(* CoDeSys 2.3.9.31 project: CL13-ARM.pro *)
(* Libraries: TcBase.lib 14.5.09 11:14:08, TcSystem.lib 27.2.12 14:08:36, TcUtilities.lib 10.1.13 19:12:12, STANDARD.LIB 5.6.98 11:03:02, TcBABasic.lib 29.10.09 13:26:44 *)

(* Task configuration *)
TASK Standard (PRIORITY := 0, INTERVAL := T#10ms);
	MAIN
END_TASK

(* Global variable list: Global_Variables *)
VAR_GLOBAL
	AllLightsOn: BOOL;
	AllLightsOff: BOOL;

	IsAllesUitInAchterbouw : BOOL; (* feedback over lichtstatus achterbouw *)
	IsAllesUitInSalon : BOOL; (* feedback over lichtstatus salon *)

	LED_Rolluik_Voorgevel_Up AT %Q*: BOOL;  (*Terugkoppeling status neersignaal*)
	LED_Rolluik_Voorgevel_Down AT %Q*: BOOL; (*Terugkoppeling status neersignaal*)

	(* Tijdsgerelateerde zaken *)
	time_RTC 				: DT;
	time_RTCEX 				: DT;
	time_RTCEX2 			: TIMESTRUCT;
	nMicroseconds 			: DWORD;

	firstCycle					: BOOL;
	status 					: StatusVariables;
	WaterTeller				:UDINT;
	AutoMode				: BOOL;
END_VAR

(* Global variable list: Input_variables *)
VAR_GLOBAL
	DK_Gang_A AT %I*: BOOL;
	DK_Gang_B AT %I*: BOOL;
	DK_Gang_C AT %I*: BOOL;
	DK_Gang_D AT %I*: BOOL;
	DK_Voordeur_BEL AT %I*: BOOL;
	DK_Toilet AT %I*:BOOL;

(* D1 / centrale kolom keuken - 1 / 6V*)
	DK_Kolom1_A  AT %I*: BOOL; (* Eiland *)
	DK_Kolom1_B  AT %I*: BOOL; (* Eettafel DIMMER *)
	DK_Kolom1_C  AT %I*: BOOL; (* Waskot *)
	DK_Kolom1_D  AT %I*: BOOL; (* Grid IN - Bureau *)
	DK_Kolom1_E  AT %I*: BOOL; (* Dampkap *)
	DK_Kolom1_F  AT %I*: BOOL; (*  *)

(* D2 / centrale kolom keuken - 2 / 4V*)
	DK_Kolom2_A  AT %I*: BOOL; (* Renson Eco *)
	DK_Kolom2_B  AT %I*: BOOL; (* Renson HDC *)
	DK_Kolom2_C  AT %I*: BOOL; (* Renson Boost/Nightcooling *)
	DK_Kolom2_D  AT %I*: BOOL; (* Renson Empty House *)

(* D3 / achtergevel - 1 / 6V*)
	DK_Achtergevel_A  AT %I*: BOOL; (* Buitenverlichting *)
	DK_Achtergevel_B  AT %I*: BOOL; (* Eettafel DIMMER *)
	DK_Achtergevel_C  AT %I*: BOOL; (* Ontbijtkast *)
	DK_Achtergevel_D  AT %I*: BOOL; (*  *)
	DK_Achtergevel_E  AT %I*: BOOL; (* Rolgordijn op *)
	DK_Achtergevel_F  AT %I*: BOOL; (* Rolgordijn neer  *)

(* D11 / Salon / 4V *)
	DK_Salon_A  AT %I*: BOOL; (* Wandlampen zetel DIMMER *)
	DK_Salon_B  AT %I*: BOOL; (*  Rolluik voorgevel *)
	DK_Salon_C  AT %I*: BOOL; (*  *)
	DK_Salon_D  AT %I*: BOOL; (*  *)

	NC_Water AT %I*:BOOL; (* NC contact Elster watermeter *)

END_VAR

(* Global variable list: Output_variables *)
VAR_GLOBAL
	L1_Oversteek 	AT %Q* 		: BOOL; 	(* Oversteek buiten *)
	L2_Eettafel		AT %Q* 		: UINT; 	(* Licht boven de eettafel *)
	L3_Bureau		AT %Q* 		: BOOL;	(* Licht bureau *)
	L4_Ontbijtkast 	AT %Q*		: BOOL;
	L5_Eiland		AT %Q* 		: BOOL; 	(* L5 - Deltalight profiel boven eiland *)
	L6_Bijkeuken		AT %Q*		: BOOL;	(* verlichting in de bijkeuken *)
	L7_Living		AT %Q* 		: BOOL; 	(* Licht living *)
	L8_Salon		AT %Q*		: UINT; 	(* Licht salon *)

	L_Gang_GLV 		AT %Q* 		: BOOL; 	(* L10 *)
	L_Toilet 			AT %Q* 		: BOOL;    (* L11 *)
	L_Kelder 		AT %Q* 		: BOOL;    (* L12_Licht kelder *)

	L2_Status 					: BOOL; 	(* Terugkoppeling van de status voor het licht boven de eettafel *)
	L8_Status 					: BOOL; 	(* Terugkoppeling van de status voor het licht in het salon *)


	HealthBox 		AT %Q* 		: BOOL; (* 230v Renson Healthbox *)
	DK_Kolom1_LED 	AT %Q* 		: BOOL;
	DK_Salon_LED 	AT %Q*		 : BOOL;
	DK_Kolom2_LED1 AT %Q*		 : BOOL;
	DK_Achtergevel_LED AT %Q* 	: BOOL;

	Auto_Rolluik_Voorgevel_Up	: BOOL;
	Auto_Rolluik_Voorgevel_Down	: BOOL;



	Rolluik_Voorgevel_Up AT %Q* : BOOL;
	Rolluik_Voorgevel_Down AT %Q* : BOOL;
	Deurbel AT %Q* : BOOL;

	M_Keuken_Op 		AT %Q* 		: BOOL;
	M_Keuken_Neer		AT %Q*		: BOOL;

(* een bit wordt geadresseerd door middel van een "Byte nr"."Bit nr"
Waarbij de byte nummer gewoon mag optellen en de bitnummer gaat van 0 tot en met 7 *)

	(*merker_OmTeTesten	AT %MX0.0 : BOOL;
	M_Licht_Eiland		AT %MX0.1 : BOOL;*)

END_VAR

(* Global variable list: PushButtons *)
VAR_GLOBAL

	Button_Kolom1_A : FB_Click;
	Button_Kolom1_C: FB_Click;
	Button_Kolom1_D: FB_Click;
	Button_Kolom1_E: FB_Click;
	Button_Kolom1_F: FB_Click;

	Click_Kolom2_A: FB_Click;
	Click_Kolom2_B: FB_Click;
	Click_Kolom2_C: FB_Click;
	Click_Kolom2_D: FB_Click;

	Click_Toilet : FB_Click;
	Click_Salon_A : FB_Click;
	Click_Salon_B : FB_Click;
	Click_Salon_C : FB_Click;
	Click_Salon_D: FB_Click;

	PushButton_Gang_A: FB_Toggle;
	PushButton_Gang_B: FB_Click;
	PushButton_Gang_C: FB_Toggle;
	PushButton_Gang_D: FB_Click;

	PushButton_Achtergevel_A : FB_Click;
	PushButton_Achtergevel_B : FB_Click;
	PushButton_Achtergevel_C: FB_Click;
	PushButton_Achtergevel_D: FB_Click;
	PushButton_Achtergevel_E: FB_Click;
	PushButton_Achtergevel_F: FB_Click;


END_VAR

(* Global variable list: TwinCAT_Configuration *)
(* Generated automatically by TwinCAT - (read only) *)
VAR_CONFIG
	.LED_Rolluik_Voorgevel_Up AT %QX4.0 : BOOL;
	.LED_Rolluik_Voorgevel_Down AT %QX4.1 : BOOL;
	.DK_Gang_A AT %IX0.0 : BOOL;	(*  ~ {LinkedWith:TIID^Device 2 (CX8000-BK)^Box 1 (CX8000-BK)^Term 2 (KL1859)^Channel 1^Input} *)
	.DK_Gang_B AT %IX0.1 : BOOL;	(*  ~ {LinkedWith:TIID^Device 2 (CX8000-BK)^Box 1 (CX8000-BK)^Term 2 (KL1859)^Channel 2^Input} *)
	.DK_Gang_C AT %IX0.2 : BOOL;	(*  ~ {LinkedWith:TIID^Device 2 (CX8000-BK)^Box 1 (CX8000-BK)^Term 2 (KL1859)^Channel 3^Input} *)
	.DK_Gang_D AT %IX0.3 : BOOL;	(*  ~ {LinkedWith:TIID^Device 2 (CX8000-BK)^Box 1 (CX8000-BK)^Term 2 (KL1859)^Channel 4^Input} *)
	.DK_Voordeur_BEL AT %IX0.4 : BOOL;	(*  ~ {LinkedWith:TIID^Device 2 (CX8000-BK)^Box 1 (CX8000-BK)^Term 2 (KL1859)^Channel 6^Input} *)
	.DK_Toilet AT %IX0.5 : BOOL;	(*  ~ {LinkedWith:TIID^Device 2 (CX8000-BK)^Box 1 (CX8000-BK)^Term 2 (KL1859)^Channel 5^Input} *)
	.DK_Kolom1_A AT %IX0.6 : BOOL;	(*  ~ {LinkedWith:TIID^Device 2 (CX8000-BK)^Box 1 (CX8000-BK)^Term 3 (KL1809)^Channel 1^Input} *)
	.DK_Kolom1_B AT %IX0.7 : BOOL;	(*  ~ {LinkedWith:TIID^Device 2 (CX8000-BK)^Box 1 (CX8000-BK)^Term 3 (KL1809)^Channel 2^Input} *)
	.DK_Kolom1_C AT %IX1.0 : BOOL;	(*  ~ {LinkedWith:TIID^Device 2 (CX8000-BK)^Box 1 (CX8000-BK)^Term 3 (KL1809)^Channel 3^Input} *)
	.DK_Kolom1_D AT %IX1.1 : BOOL;	(*  ~ {LinkedWith:TIID^Device 2 (CX8000-BK)^Box 1 (CX8000-BK)^Term 3 (KL1809)^Channel 4^Input} *)
	.DK_Kolom1_E AT %IX1.2 : BOOL;	(*  ~ {LinkedWith:TIID^Device 2 (CX8000-BK)^Box 1 (CX8000-BK)^Term 3 (KL1809)^Channel 5^Input} *)
	.DK_Kolom1_F AT %IX1.3 : BOOL;	(*  ~ {LinkedWith:TIID^Device 2 (CX8000-BK)^Box 1 (CX8000-BK)^Term 3 (KL1809)^Channel 6^Input} *)
	.DK_Kolom2_A AT %IX1.4 : BOOL;
	.DK_Kolom2_B AT %IX1.5 : BOOL;
	.DK_Kolom2_C AT %IX1.6 : BOOL;
	.DK_Kolom2_D AT %IX1.7 : BOOL;
	.DK_Achtergevel_A AT %IX8.0 : BOOL;	(*  ~ {LinkedWith:TIID^Device 2 (CX8000-BK)^Box 1 (CX8000-BK)^Term 3 (KL1809)^Channel 11^Input} *)
	.DK_Achtergevel_B AT %IX8.1 : BOOL;	(*  ~ {LinkedWith:TIID^Device 2 (CX8000-BK)^Box 1 (CX8000-BK)^Term 3 (KL1809)^Channel 12^Input} *)
	.DK_Achtergevel_C AT %IX8.2 : BOOL;	(*  ~ {LinkedWith:TIID^Device 2 (CX8000-BK)^Box 1 (CX8000-BK)^Term 3 (KL1809)^Channel 13^Input} *)
	.DK_Achtergevel_D AT %IX8.3 : BOOL;	(*  ~ {LinkedWith:TIID^Device 2 (CX8000-BK)^Box 1 (CX8000-BK)^Term 3 (KL1809)^Channel 14^Input} *)
	.DK_Achtergevel_E AT %IX8.4 : BOOL;	(*  ~ {LinkedWith:TIID^Device 2 (CX8000-BK)^Box 1 (CX8000-BK)^Term 3 (KL1809)^Channel 15^Input} *)
	.DK_Achtergevel_F AT %IX8.5 : BOOL;	(*  ~ {LinkedWith:TIID^Device 2 (CX8000-BK)^Box 1 (CX8000-BK)^Term 3 (KL1809)^Channel 16^Input} *)
	.DK_Salon_A AT %IX2.0 : BOOL;	(*  ~ {LinkedWith:TIID^Device 2 (CX8000-BK)^Box 1 (CX8000-BK)^Term 3 (KL1809)^Channel 7^Input} *)
	.DK_Salon_B AT %IX2.1 : BOOL;	(*  ~ {LinkedWith:TIID^Device 2 (CX8000-BK)^Box 1 (CX8000-BK)^Term 3 (KL1809)^Channel 8^Input} *)
	.DK_Salon_C AT %IX2.2 : BOOL;	(*  ~ {LinkedWith:TIID^Device 2 (CX8000-BK)^Box 1 (CX8000-BK)^Term 3 (KL1809)^Channel 9^Input} *)
	.DK_Salon_D AT %IX2.3 : BOOL;	(*  ~ {LinkedWith:TIID^Device 2 (CX8000-BK)^Box 1 (CX8000-BK)^Term 3 (KL1809)^Channel 10^Input} *)
	.NC_Water AT %IX4.0 : BOOL;	(*  ~ {LinkedWith:TIID^Device 2 (CX8000-BK)^Box 1 (CX8000-BK)^Term 5 (KL1809)^Channel 1^Input} *)
	.L1_Oversteek AT %QX20.0 : BOOL;	(*  ~ {LinkedWith:TIID^Device 2 (CX8000-BK)^Box 1 (CX8000-BK)^Term 6 (KL2809)^Channel 1^Output} *)
	.L2_Eettafel AT %QB16 : UINT;	(*  ~ {LinkedWith:TIID^Device 2 (CX8000-BK)^Box 1 (CX8000-BK)^Term 13 (KL2751)^Channel 1^Data Out} *)
	.L3_Bureau AT %QX20.1 : BOOL;	(*  ~ {LinkedWith:TIID^Device 2 (CX8000-BK)^Box 1 (CX8000-BK)^Term 6 (KL2809)^Channel 2^Output} *)
	.L4_Ontbijtkast AT %QX20.2 : BOOL;
	.L5_Eiland AT %QX20.3 : BOOL;
	.L6_Bijkeuken AT %QX20.4 : BOOL;
	.L7_Living AT %QX20.5 : BOOL;
	.L8_Salon AT %QB18 : UINT;	(*  ~ {LinkedWith:TIID^Device 2 (CX8000-BK)^Box 1 (CX8000-BK)^Term 14 (KL2751)^Channel 1^Data Out} *)
	.L_Gang_GLV AT %QX4.5 : BOOL;	(*  ~ {LinkedWith:TIID^Device 2 (CX8000-BK)^Box 1 (CX8000-BK)^Term 6 (KL2809)^Channel 14^Output} *)
	.L_Toilet AT %QX4.6 : BOOL;	(*  ~ {LinkedWith:TIID^Device 2 (CX8000-BK)^Box 1 (CX8000-BK)^Term 6 (KL2809)^Channel 13^Output} *)
	.L_Kelder AT %QX4.4 : BOOL;	(*  ~ {LinkedWith:TIID^Device 2 (CX8000-BK)^Box 1 (CX8000-BK)^Term 6 (KL2809)^Channel 16^Output} *)
	.HealthBox AT %QX5.5 : BOOL;	(*  ~ {LinkedWith:TIID^Device 2 (CX8000-BK)^Box 1 (CX8000-BK)^Term 2 (KL1859)^Channel 8^Output} *)
	.DK_Kolom1_LED AT %QX5.6 : BOOL;	(*  ~ {LinkedWith:TIID^Device 2 (CX8000-BK)^Box 1 (CX8000-BK)^Term 7 (KL2809)^Channel 2^Output} *)
	.DK_Salon_LED AT %QX5.7 : BOOL;	(*  ~ {LinkedWith:TIID^Device 2 (CX8000-BK)^Box 1 (CX8000-BK)^Term 7 (KL2809)^Channel 1^Output} *)
	.DK_Kolom2_LED1 AT %QX6.0 : BOOL;
	.DK_Achtergevel_LED AT %QX20.6 : BOOL;
	.Rolluik_Voorgevel_Up AT %QX5.0 : BOOL;	(*  ~ {LinkedWith:TIID^Device 2 (CX8000-BK)^Box 1 (CX8000-BK)^Term 8 (KL2012)^Channel 1^Output} *)
	.Rolluik_Voorgevel_Down AT %QX5.1 : BOOL;	(*  ~ {LinkedWith:TIID^Device 2 (CX8000-BK)^Box 1 (CX8000-BK)^Term 8 (KL2012)^Channel 2^Output} *)
	.Deurbel AT %QX5.2 : BOOL;	(*  ~ {LinkedWith:TIID^Device 2 (CX8000-BK)^Box 1 (CX8000-BK)^Term 2 (KL1859)^Channel 4^Output} *)
	.M_Keuken_Op AT %QX12.1 : BOOL;	(*  ~ {LinkedWith:TIID^Device 2 (CX8000-BK)^Box 1 (CX8000-BK)^Term 9 (KL2012)^Channel 1^Output} *)
	.M_Keuken_Neer AT %QX12.2 : BOOL;	(*  ~ {LinkedWith:TIID^Device 2 (CX8000-BK)^Box 1 (CX8000-BK)^Term 9 (KL2012)^Channel 2^Output} *)
END_VAR

(* Global variable list: Visualisation_variables *)
VAR_GLOBAL

	Visu_Licht_Oversteek		AT %MX0.0 			: BOOL;
	Visu_Dimmer_Eettafel		AT %MX0.1 			: BOOL;
	Visu_L3 					AT %MX0.2			: BOOL; (* Licht bureau *)
	Visu_Ontbijtkast 			AT %MX0.3			: BOOL;
	Visu_Eiland				AT %MX0.4			: BOOL;
	Visu_Bijkeuken			AT %MX0.5			: BOOL;
	Visu_Licht_Living 			AT %MX0.6			: BOOL;
	Visu_Dimmer_Salon 		AT %MX0.7 			: BOOL;

	Visu_Salon_TV			AT %MX0.8			: BOOL; (* Nog niet in gebruik *)
	Visu_Licht_Gang			AT %MX0.9			: BOOL; (* L10 *)
	Visu_Licht_Toilet 			AT %MX0.10			: BOOL; (* L11 *)
	Visu_Licht_Kelder			AT %MX0.11			: BOOL; (* L12 *)

	(* Andere lichten komen hier *)

	Visu_Rolluik_Voorgevel_Up	AT %MX2.0	 	: BOOL;
	Visu_Rolluik_Voorgevel_Down	AT %MX2.1	 	: BOOL;
	Visu_Rolgordijn_Up			AT %MX2.3		: BOOL;
	Visu_Rolgordijn_Neer			AT %MX2.4		: BOOL;
	Visu_AllesUit 					AT %MX2.5		: BOOL;

	Visu_Deurbel 				: BOOL;
	Visu_AllesAan 				: BOOL;
	Visu_HEALTHBOX			: BOOL; (* Healthbox *)
	Visu_Dimmer_Salon_Status		: REAL;
	Visu_Dimmer_Eettafel_Status	: REAL;

	Visu_Sfeer_Avond				: BOOL;
	Visu_AutoMode				: BOOL;


(* alle types die op een byte grootte hebben, woorden weergegeven zoals:
	MerkerByte_2		AT %MB2 : BYTE;
	MerkerByte_3		AT %MB3 : BYTE;
	MerkerByte_4		AT %MB4 : BYTE;
	MerkerByte_5		AT %MB5 : BYTE;

(* alle types die op een woord grootte hebben, woorden weergegeven zoals: *)
	MerkerWoord_10		AT %MW10 : INT;
	MerkerWoord_12		AT %MW12 : UINT;
	MerkerWoord_14		AT %MW14 : INT;
	MerkerWoord_16		AT %MW16 : UINT;

(* alle types die op een dubbelwoord grootte hebben, woorden weergegeven zoals: *)
	MerkerDWoord_20		AT %MD20 : DINT;
	MerkerDWoord_24		AT %MD24 : UDINT;
	MerkerDWoord_28		AT %MD28 : REAL;
	MerkerDWoord_32		AT %MD32 : UINT;

*)


END_VAR

(* Data type *)
TYPE StatusVariables :
STRUCT

END_STRUCT
END_TYPE

(* POU MAIN, ST *)
PROGRAM MAIN
VAR
END_VAR
Process_Inputs;
Rolluiken;
Deurbel_Programma;
Dimmers;
Control_Lights_ST;
Ventilation;
BezorgFeedbackAanLeds;
PRG_Clock;
MAIN_1;

firstCycle := Systemtaskinfoarr[1].firstCycle;
(*SetStatusStruct; *)
Smartmeters;
ResetInputs;
END_PROGRAM

(* POU Process_Inputs, ST *)
PROGRAM Process_Inputs
VAR
	R_Trig_AllesUit: R_TRIG;
END_VAR
PushButton_Gang_B(ingang:= DK_Gang_B); (* linkt de fysieke input aan de functie block FB_Click *)
PushButton_Gang_D(ingang:= DK_Gang_D);
Button_Kolom1_A(ingang:= DK_Kolom1_A);
Button_Kolom1_C(ingang:= DK_Kolom1_C);
Button_Kolom1_D(ingang:= DK_Kolom1_D);
Button_Kolom1_E(ingang:= DK_Kolom1_E);
Button_Kolom1_F(ingang:= DK_Kolom1_F);
Click_Toilet(ingang:= DK_Toilet);

Click_Kolom2_A(ingang := DK_Kolom2_A);
Click_Kolom2_B(ingang := DK_Kolom2_B);
Click_Kolom2_C(ingang := DK_Kolom2_C);
Click_Kolom2_D(ingang := DK_Kolom2_D);

PushButton_Achtergevel_A(ingang:= DK_Achtergevel_A);
PushButton_Achtergevel_B(ingang:= DK_Achtergevel_B);
PushButton_Achtergevel_C(ingang:= DK_Achtergevel_C);
PushButton_Achtergevel_D(ingang:= DK_Achtergevel_D);
PushButton_Achtergevel_E(ingang:= DK_Achtergevel_E);
PushButton_Achtergevel_F(ingang:= DK_Achtergevel_F);

AllLightsOff := Visu_AllesUit OR PushButton_Gang_D.LangClick;
AllLightsOn := Visu_AllesAan OR PushButton_Gang_D.TweeClick;
END_PROGRAM

(* POU Rolluiken, ST *)
PROGRAM Rolluiken
VAR
	Rolluik_Voorgevel: Rolluik;
	Rolgordijn_Keuken: Rolluik;
END_VAR
Rolgordijn_Keuken
(
	DrukknopOp:=  PushButton_Achtergevel_D.EenClick OR Visu_Rolgordijn_Up,
	DrukknopNeer:= PushButton_Achtergevel_C.EenClick OR Visu_Rolgordijn_Neer,
	Tijd:= t#100s,
	UitgOp=> M_Keuken_Op,
	UitgNeer=>M_Keuken_Neer );

Rolluik_Voorgevel
(
	DrukknopOp:=  Button_Kolom1_D.EenClick OR Visu_Rolluik_Voorgevel_Up OR Click_Salon_D.EenClick,
	DrukknopNeer:= Button_Kolom1_C.EenClick OR Visu_Rolluik_Voorgevel_Down OR Click_Salon_C.TweeClick,
	Tijd:= t#20s,
	UitgOp=> Rolluik_Voorgevel_Up,
	UitgNeer=>Rolluik_Voorgevel_Down );
END_PROGRAM

(* POU TestCode/Rolluik, ST *)
FUNCTION_BLOCK Rolluik
VAR_INPUT
	DrukknopOp: BOOL;
	DrukknopNeer: BOOL;
	Tijd: TIME := t#20s;
END_VAR
VAR_OUTPUT
	UitgOp: BOOL;
	UitgNeer: BOOL;
END_VAR
VAR
	Stap: INT;
	TimerOp: TON;
	TimerNeer: TON;
	rDrukknopOp: R_TRIG;
	rDrukknopNeer: R_TRIG;
END_VAR
TimerOp(IN:= Stap = 10 , PT:= Tijd , Q=> , ET=> );
TimerNeer(IN:= Stap = 20 , PT:= Tijd , Q=> , ET=> );

rDrukknopOp(CLK:= DrukknopOp , Q=> );
rDrukknopNeer(CLK:= DrukknopNeer , Q=> );

CASE Stap OF

0:
	IF rDrukknopOp.Q THEN
		Stap := 10;
	END_IF

	IF rDrukknopNeer.Q THEN
		Stap := 20;
	END_IF

10:
	IF DrukknopNeer OR TimerOp.Q  THEN
		Stap := 0;
	END_IF

20:

	IF DrukknopOp OR TimerNeer.Q THEN
		Stap := 0;
	END_IF

END_CASE


UitgOp := Stap = 10;
UitgNeer := Stap = 20;
END_FUNCTION_BLOCK

(* POU Deurbel_Programma, LD *)
PROGRAM Deurbel_Programma
VAR
	Timer_Deurbel: TOF;
	Status_Deurbel: BOOL;
END_VAR
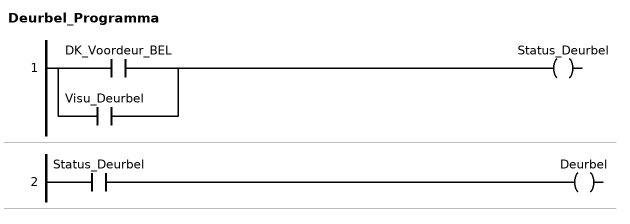
_LD_ (* Ladder Diagram *)
NETWORK 1
	{ [DK_Voordeur_BEL] | [Visu_Deurbel] } --- (Status_Deurbel)
NETWORK 2
	[Status_Deurbel] --- (Deurbel)
_END_LD_
(* the same logic as Structured Text *)
(* Network 1 *)
Status_Deurbel := DK_Voordeur_BEL OR Visu_Deurbel;
(* Network 2 *)
Deurbel := Status_Deurbel;
END_PROGRAM

(* POU Dimmers, ST *)
PROGRAM Dimmers
VAR
	Dimmer_Eettafel: FB_Dimmer1SwitchEco;
	(*Dimmer_Eettafel2: FB_Dimmer1Switch;*)
	Dimmer_SalonL9: FB_Dimmer1SwitchEco;
END_VAR
Dimmer_Eettafel
(
bSwitchDimm:= Visu_Dimmer_Eettafel OR PushButton_Gang_B.TweeClick OR DK_Kolom1_B,
tDimmTime:= t#3s,
bOn:= AllLightsOn,
bOff:= AllLightsOff,
nOut=>L2_Eettafel,
bLight => L2_Status,
);

Visu_Dimmer_Salon_Status := OnAScaleOfZeroToTen(L8_Salon);
Visu_Dimmer_Eettafel_Status := OnAScaleOfZeroToTen(L2_Eettafel);

Dimmer_SalonL9
(
	bSwitchDimm:= DK_Salon_A OR Visu_Dimmer_Salon,
	bOn:= AllLightsOn,
	bOff:= AllLightsOff,
	tSwitchOverTime:= ,
	tDimmTime:= t#3s,

	nOut=>L8_Salon ,
	bLight=>L8_Status );
END_PROGRAM

(* POU Functions/OnAScaleOfZeroToTen, ST *)
FUNCTION OnAScaleOfZeroToTen : LREAL
VAR_INPUT
	ValueIn : INT;

END_VAR
VAR
END_VAR
OnAScaleOfZeroToTen := ValueIn /  3267.6;
END_FUNCTION

(* POU Control_Lights_ST, ST *)
PROGRAM Control_Lights_ST
VAR
	FB_Light_Hallway_Downstairs: FB_Light;
	FB_Light_Toilet: FB_Light;
	FB_Light_3: FB_Light;
	FB_Light_Oversteek: FB_Light;
	FB_Light_Ontbijtkast: FB_Light;
	FB_Light_Eiland : FB_Light;
	FB_Light_Kelder : FB_Light;
	FB_Light_Wasplaats : FB_Light;
	FB_Sfeer_Avond_Salon : FB_Sfeer;

	FB_Light_Living: FB_Light;
	FB_Auto_Mode: FB_Light;
END_VAR
FB_Light_Hallway_Downstairs(
	bOn:= AllLightsOn ,
	bOff:=AllLightsOff ,
	bToggle:= Visu_Licht_Gang OR DK_Gang_C
	 , bLight=> L_Gang_GLV);

FB_Auto_Mode(
	bOn:= 0 ,
	bOff:=0 ,
	bToggle:=Click_Toilet.LangClick OR Visu_AutoMode
	 , bLight=> AutoMode);

FB_Light_Toilet(
	bOn:= 0 ,
	bOff:=AllLightsOff ,
	bToggle:=Visu_Licht_Toilet OR Click_Toilet.EenClick
	 , bLight=> L_Toilet);

FB_Light_3(
	bOn:= AllLightsOn ,
	bOff:=AllLightsOff ,
	bToggle:=Button_Kolom1_A.TweeClick OR Visu_L3
	 , bLight=> L3_Bureau);

FB_Light_Oversteek(
	bOn:= 0 ,
	bOff:=AllLightsOff ,
	bToggle:=Visu_Licht_Oversteek OR PushButton_Achtergevel_A.EenClick
	 , bLight=> L1_Oversteek);

FB_Light_Ontbijtkast(
	bOn := AllLightsOn,
	bOff := AllLightsOff,
	bToggle := PushButton_Achtergevel_B.EenClick OR Visu_Ontbijtkast,
	bLight => L4_Ontbijtkast);

FB_Light_Eiland(
	bOn := AllLightsOn,
	bOff := AllLightsOff,
	bToggle := Button_Kolom1_A.EenClick OR Visu_Eiland,
	bLight => L5_Eiland);

FB_Light_Kelder(
	bOn := 0,
	bOff := AllLightsOff,
	bToggle := PushButton_Gang_B.EenClick OR Visu_Licht_Kelder,
	bLight => L_Kelder);


FB_Light_Wasplaats(
	bOn := AllLightsOn,
	bOff := AllLightsOff,
	bToggle := Button_Kolom1_E.EenClick OR Visu_Bijkeuken,
	bLight => L6_Bijkeuken);

FB_Light_Living
(
	bOn :=AllLightsOn,
	bOff := AllLightsOff,
	bToggle := Button_Kolom1_F.EenClick OR Visu_Licht_Living,
	bLight => L7_Living);

(* FB_Sfeer_Avond_Salon(Trigger:= Visu_Sfeer_Avond, default:= 0, Uitgang => L3_Bureau);*)
END_PROGRAM

(* POU TestCode/FB_Sfeer, ST *)
FUNCTION_BLOCK FB_Sfeer
VAR_INPUT
	Trigger : BOOL;
	default: BOOL;
END_VAR
VAR_OUTPUT
	Uitgang : BOOL;
END_VAR
VAR
	Getriggerd: R_TRIG;
	DoUwDing: BOOL;
END_VAR
Getriggerd(CLK:= Trigger, Q => DoUwDing);

IF DoUwDing THEN
	Uitgang := default;
END_IF
END_FUNCTION_BLOCK

(* POU Ventilation, ST *)
PROGRAM Ventilation
VAR
	FB_Ventilation_OnOff: FB_Light;
END_VAR
FB_Ventilation_OnOff(
	bOn:= 0 ,
	bOff:=0 ,
	bToggle:= Visu_HealthBox OR Button_Kolom1_E.LangClick
	 , bLight=> HealthBox);
END_PROGRAM

(* POU BezorgFeedbackAanLeds, ST *)
PROGRAM BezorgFeedbackAanLeds
VAR
END_VAR
DK_Kolom1_LED :=	NOT L5_Eiland
					AND NOT L2_Status
					AND NOT L3_Bureau
					AND NOT AutoMode;

DK_Achtergevel_LED := DK_Kolom1_LED;

DK_Salon_LED := 		NOT L8_Status AND NOT AutoMode;

DK_Kolom2_LED1 := HealthBox;
END_PROGRAM

(* POU PRG_Clock, ST *)
PROGRAM PRG_Clock
VAR
	NT_GetTime_CX				: NT_GetTime;
	GetTime						: DT;
	Clock						: RTC;

	PC_Clock_Valid				: BOOL;
	RTC_Clock_Valid				: BOOL;

	Actual_Time 					: TOD;
	Actual_Date 					: DATE;

	Actual_Date_Time				: STRING;

	Actual_Hour					: WORD;
	Actual_Minute					: WORD;
	Actual_Second				: WORD;
	Actual_Year					: WORD;
	Actual_Month					: WORD;
	Actual_Day					: WORD;
END_VAR
(* Bios time and date from PC or CX *)
NT_GetTime_CX(
	NETID		:= 	'200.255.255.154.1.1',									(* AMS NetID from PC or CX, empty string is lokal *)
	START		:= 	SystemTaskInfoArr[1].firstCycle OR						(* Update after start Runtime *)
					(DT_TO_TOD(Clock.CDT)=TOD#00:00:00) OR				(* Update if 'Clock' empty *)
					MID(DT_TO_STRING(Clock.CDT),2,21)='00',				(* Update each minute *)
	TMOUT		:= 	t#1s ,
	 );

PC_Clock_Valid 	:= NOT NT_GetTime_CX.BUSY AND NOT NT_GetTime_CX.START;

(* Time from external device *)
IF PC_Clock_Valid THEN
	GetTime := SYSTEMTIME_TO_DT(NT_GetTime_CX.TIMESTR);
END_IF

Clock(																	(* Internal clock, independent with Windows clock *)
	EN			:= PC_Clock_Valid,
	PDT		:= GetTime
	 );

RTC_Clock_Valid	:= Clock.Q;

(* Date en Time *)
IF RTC_Clock_Valid THEN
	Actual_Time 				:= DT_TO_TOD(Clock.CDT);
	Actual_Date				:= DT_TO_DATE(Clock.CDT);

	Actual_Date_Time			:= DT_TO_STRING(Clock.CDT);

	Actual_Hour 				:= STRING_TO_INT(MID(Actual_Date_Time,2,15));
	Actual_Minute 			:= STRING_TO_INT(MID(Actual_Date_Time,2,18));
	Actual_Second 			:= STRING_TO_INT(MID(Actual_Date_Time,2,21));
	Actual_Year 				:= STRING_TO_INT(MID(Actual_Date_Time,4,4));
	Actual_Month 				:= STRING_TO_INT(MID(Actual_Date_Time,2,9));
	Actual_Day 				:= STRING_TO_INT(MID(Actual_Date_Time,2,12));
END_IF
END_PROGRAM

(* POU MAIN_1, ST *)
PROGRAM MAIN_1
VAR
	CurrentTime			: TOD;
	tRolluikOp			: TOD;
	tRolluikNeer			: TOD;
	tLightGangAan		: TOD;
	tLightGangUit			: TOD;

	tLichtGangAan: TOD;
	tLichtGangUit: TOD;
	tTestAan: TOD;
	tTestUit: TOD;
	strTime: STRING;
END_VAR
P_RTC_ST;

(* dsjkfsjlqfs *)
IF firstCycle	THEN

	tRolluikOp := TOD#07:30:00;
	tRolluikNeer := TOD#17:48:30;

	tLichtGangAan:= TOD#21:04:00;
	tLichtGangUit:= TOD#22:43:00;

	tTestAan	:= TOD#00:00:00;
	tTestUit:= TOD#08:00:00;

END_IF

	tRolluikOp := TOD#07:30:00;
	tRolluikNeer := TOD#17:48:30;

	tLichtGangAan:= TOD#21:04:00;
	tLichtGangUit:= TOD#22:43:00;

	tTestAan	:= TOD#23:58:00;
	tTestUit:= TOD#23:59:00;

CurrentTime := DT_TO_TOD(time_RTC);
strTime := TOD_TO_STRING(CurrentTime);

IF AutoMode THEN
	IF CurrentTime > tRolluikOp AND CurrentTime < tRolluikNeer  THEN
	Rolluik_Voorgevel_Up := TRUE;
	Rolluik_Voorgevel_Down := FALSE;
	ELSE
	Rolluik_Voorgevel_Up := FALSE;
	Rolluik_Voorgevel_Down := TRUE;
	END_IF

	IF CurrentTime > tLichtGangAan AND CurrentTime < tLichtGangUit THEN
	L_Gang_GLV := TRUE;
	ELSE
	L_Gang_GLV := FALSE;
	END_IF
ELSE
;
	(*Rolluik_Voorgevel_Up := FALSE;
	Rolluik_Voorgevel_Down := FALSE;*)
END_IF


(*IF CurrentTime > tTestAan AND CurrentTime < tTestUit THEN
HealthBox := TRUE;
ELSE
HealthBox := FALSE;
END_IF*)
END_PROGRAM

(* POU tcUtilities/Converting/Formatting/P_RTC_ST, ST *)
PROGRAM P_RTC_ST
VAR
	syncTimer 				: TON;
	fbGetLocalTime 			: NT_GetTime;
	syncTrigger 			: F_TRIG;
	bBusy 					: BOOL;
	bError 					: BOOL;
	nErrID 					: UDINT;
	presetTime 				: TIMESTRUCT;

	fbRTC 					: RTC;
	bValid_RTC 				: BOOL;

	fbRTC_EX 				: RTC_EX;
	bValid_RTCEX 			: BOOL;
	nMilliseconds 			: DWORD;

	fbRTC_EX2 				: RTC_EX2;
	bValid_RTCEX2 			: BOOL;

END_VAR
syncTimer(
	IN			:= NOT syncTimer.q,
	PT			:= T#5s,
	Q			=> ,
	ET			=> );

fbGetLocalTime(
	NETID		:= ,
	START		:= syncTimer.Q	OR systemtaskinfoarr[1].firstCycle,
	TMOUT		:= ,
	BUSY		=> ,
	ERR		=> bError,
	ERRID		=> nErrID,
	TIMESTR	=> presetTime);

syncTrigger(
	CLK			:= fbGetLocalTime.BUSY AND NOT bError,
	Q=> 			);

fbRTC(
	EN			:= syncTrigger.Q,
	PDT		:= SYSTEMTIME_TO_DT(presetTime),
	Q			=> bValid_RTC,
	CDT=> 		time_RTC);

fbRTC_EX(
	EN			:= syncTrigger.Q,
	PDT		:= SYSTEMTIME_TO_DT(presetTime),
	PMSEK		:= presetTime.wMilliseconds,
	Q			=> bValid_RTCEX,
	CDT		=> time_RTCEX,
	CMSEK		=> nMilliseconds);

fbRTC_EX2(
	EN			:= syncTrigger.Q,
	PDT		:= presetTime,
	PMICRO		:= 0,
	Q			=> bValid_RTCEX2,
	CDT		=> time_RTCEX2,
	CMICRO		=> nMicroseconds);
END_PROGRAM

(* POU Smartmeters, ST *)
PROGRAM Smartmeters
VAR
	fet_pulse		: F_TRIG;
	pulse		: BOOL;
	NoChange	: BOOL;
END_VAR
VAR RETAIN PERSISTENT
	teller		: UDINT;
END_VAR
NoChange:= NC_Water;

IF NoChange = TRUE THEN
	pulse:= FALSE;
END_IF

fet_pulse(clk:=NC_Water);
pulse := fet_pulse.Q;

IF pulse THEN
	teller:= teller + 1;
END_IF

WaterTeller:=teller;
END_PROGRAM

(* POU ResetInputs, ST *)
PROGRAM ResetInputs
VAR
	Tap_Ontbijtkast : Tap;
	Tap_AllesUit : Tap;
	Tap_GangBeneden : Tap;
END_VAR
Tap_Ontbijtkast(trigger:=Visu_Ontbijtkast);
Tap_GangBeneden(trigger := Visu_Licht_Gang);
Tap_AllesUit(trigger := Visu_AllesUit);
END_PROGRAM

(* POU TestCode/Tap, ST *)
FUNCTION_BLOCK Tap
VAR_INPUT
	trigger : BOOL;
END_VAR
VAR_OUTPUT
END_VAR
VAR
	Detect: R_TRIG;
	WasPressed : BOOL;
END_VAR
Detect(CLK:=trigger , Q=>WasPressed);

IF WasPressed THEN
	trigger := FALSE;
END_IF
END_FUNCTION_BLOCK

(* POU SetStatusStruct, ST *)
PROGRAM SetStatusStruct
VAR
END_VAR
(*status.L_Eiland := L5_Eiland;
status.L7_Living:= L7_Living;
status.Deurbel:= Deurbel;
status.HealthBox:= HealthBox;
status.L_2Status := L_2Status;
status.L_2Value := L2_Eettafel;
status.L3_Bureau:= L3_Bureau;
status.L8_Salon:= L8_Salon;
status.L_9Status:= L_9Status;
status.L_Eiland:= L5_Eiland;
status.L_Gang_GLV := L_Gang_GLV;
status.L_Kelder:= L_Kelder;
status.L7_Living:= L7_Living;
status.L1_Oversteek := L1_Oversteek;
status.L_Toilet := L_Toilet;
status.Rolluik_Voorgevel_Down:= Rolluik_Voorgevel_Down;
status.Rolluik_Voorgevel_Up:= Rolluik_Voorgevel_Up; *)
;
END_PROGRAM

(* POU Function Blocks/FB_Click, ST *)
FUNCTION_BLOCK FB_Click
VAR_INPUT
	Ingang				: BOOL;
END_VAR
VAR_OUTPUT
	NoChange			:BOOL;
	EenClick				: BOOL;
	TweeClick			: BOOL;
	DrieClick				: BOOL;
	LangClick			: BOOL;
END_VAR
VAR
	RisingEdgeIngang	: R_TRIG;
	FalingEdgeTimer1	: F_TRIG;
	Timer1				: TOF;
	teller				: UINT;
END_VAR
NoChange := Ingang;
IF ingang = FALSE THEN
	EenClick:= FALSE;
	TweeClick:= FALSE;
	DrieClick:= FALSE;
	LangClick:= FALSE;
END_IF;

RisingEdgeIngang(CLK:=Ingang);
Timer1(IN:= RisingEdgeIngang.Q, PT:= T#400ms);
FalingEdgeTimer1(CLK:=Timer1.Q );

IF RisingEdgeIngang.Q THEN
	teller := teller +1;
END_IF

IF FalingEdgeTimer1.Q THEN
	IF ingang THEN
		LangClick := TRUE;
	ELSE
		CASE teller OF
			1: EenClick:= TRUE;
			2: TweeClick:= TRUE;
			3: DrieClick:= TRUE;
		END_CASE
	END_IF
	teller := 0;
END_IF
END_FUNCTION_BLOCK

(* POU Function Blocks/FB_LightControl_Local, ST *)
FUNCTION_BLOCK FB_LightControl_Local
VAR_INPUT
	TOGGLE: BOOL;
	Set: BOOL;
	Reset: BOOL;
	ForceerAan: BOOL;
	ForceerUit: BOOL;
	TijdAutoUit: TIME;
END_VAR
VAR_OUTPUT
	uitgang: BOOL;
END_VAR
VAR
	Licht: BOOL;
	RisingEdgeToggle: R_TRIG;
	Timer1: TON;
	RisingEdgeReset: R_TRIG;
	RisingEdgeSet: R_TRIG;
END_VAR
(*====TOGGLE AAN/UIT ==================================*)
(*Toggle licht aan / uit*)
RisingEdgeToggle(CLK := Toggle );
IF (RisingEdgeToggle.Q) THEN
	Licht := NOT Licht;
END_IF


(*====AUTOMATISCH UIT OP TIJD==========================*)
Timer1(IN:= Licht AND TijdAutoUit <> T#0s, PT:= TijdAutoUit );
IF Timer1.Q THEN
	licht := FALSE;
END_IF

(*====SET/RESET===================================*)
RisingEdgeSet(CLK := Set );
IF (RisingEdgeSet.Q) THEN
	Licht := TRUE;
END_IF
RisingEdgeReset(CLK := Reset );
IF (RisingEdgeReset.Q) THEN
	Licht := FALSE;
END_IF

(*====Forceer aan/uit======================================*)
uitgang := NOT(ForceerUit) AND (ForceerAan OR Licht);
END_FUNCTION_BLOCK

(* POU Function Blocks/FB_Toggle, LD *)
FUNCTION_BLOCK FB_Toggle
VAR_INPUT
	iToggle: BOOL;
END_VAR
VAR_OUTPUT
	oUitgang : BOOL;
END_VAR
VAR
	status: BOOL;
	RisingEdge: R_TRIG;
END_VAR
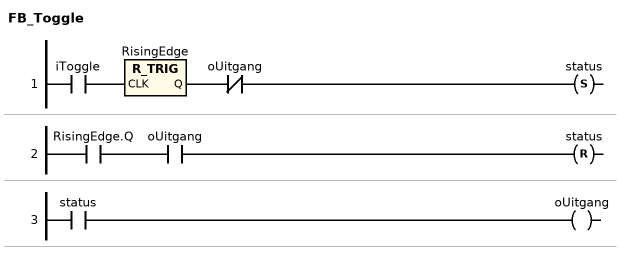
_LD_ (* Ladder Diagram *)
NETWORK 1
	[iToggle] - RisingEdge:R_TRIG(CLK: *) - [/oUitgang] --- (S status)
NETWORK 2
	[RisingEdge.Q] - [oUitgang] --- (R status)
NETWORK 3
	[status] --- (oUitgang)
_END_LD_
(* the same logic as Structured Text *)
(* Network 1 *)
RisingEdge(CLK := iToggle);
IF RisingEdge.Q AND NOT oUitgang THEN status := TRUE; END_IF;
(* Network 2 *)
IF RisingEdge.Q AND oUitgang THEN status := FALSE; END_IF;
(* Network 3 *)
oUitgang := status;
END_FUNCTION_BLOCK

(* Visualisation TC_VISU
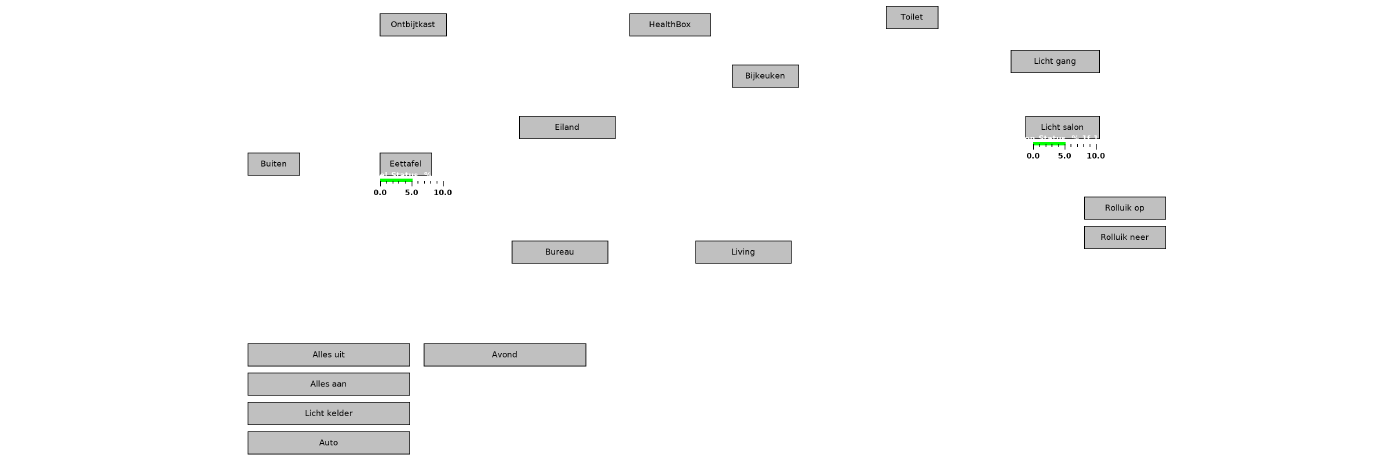
rounded rectangle at (220,240)-(291,271): text "Eettafel"; alarm colour if .L2_Status; taps .Visu_Dimmer_Eettafel
rounded rectangle at (1080,100)-(1201,131): text "Licht gang"; alarm colour if .L_Gang_GLV; taps .Visu_Licht_Gang
rounded rectangle at (410,190)-(541,221): text "Eiland"; alarm colour if .L5_Eiland; taps .Visu_Licht_Beneden
rounded rectangle at (910,40)-(981,71): text "Toilet"; alarm colour if .L_Toilet; taps .Visu_Licht_Toilet
rounded rectangle at (40,580)-(261,611): text "Licht kelder"; alarm colour if .L_Kelder; taps .Visu_Licht_Kelder
rounded rectangle at (40,500)-(261,531): text "Alles uit"; alarm colour if .AllLightsOff; taps .Visu_AllesUit
rounded rectangle at (1100,190)-(1201,221): text "Licht salon"; alarm colour if .L8_Status; taps .Visu_Dimmer_Salon
rounded rectangle at (40,540)-(261,571): text "Alles aan"; alarm colour if .AllLightsOn; taps .Visu_AllesAan
group at (1100,220)-(1211,251)
  rectangle at (5,0)-(6,1): text "{ExtendedElement},Visu\ElementDLL.ete,1,@Bargraph,111,31,0,0,0,Visu_Dimmer_Salon_Status,,%.1f,1,5,0,10,0,0,0,0,0,0,0,-13,16,700,Arial,0,255,0,255,0,0,0,0,0,0,0,0,0,,0,"
  rectangle at (12,5)-(61,9): alarm colour if (Visu_Dimmer_Salon_Status) < 0; right ((Visu_Dimmer_Salon_Status * 1.0) - 5)  * 9.6
  rectangle at (0,16)-(24,28): text "0.0"
  rectangle at (48,16)-(72,28): text "5.0"
  rectangle at (91,16)-(124,28): text "10.0"
group at (210,270)-(321,301)
  rectangle at (5,0)-(6,1): text "{ExtendedElement},Visu\ElementDLL.ete,1,@Bargraph,111,31,0,0,0,Visu_Dimmer_Eettafel_Status,,%.1f,1,5,0,10,0,0,0,0,0,0,0,-13,16,700,Arial,0,255,0,255,0,0,0,0,0,0,0,0,0,,0,"
  rectangle at (12,5)-(61,9): alarm colour if (Visu_Dimmer_Eettafel_Status) < 0; right ((Visu_Dimmer_Eettafel_Status * 1.0) - 5)  * 9.6
  rectangle at (0,16)-(24,28): text "0.0"
  rectangle at (48,16)-(72,28): text "5.0"
  rectangle at (91,16)-(124,28): text "10.0"
rounded rectangle at (400,360)-(531,391): text "Bureau"; alarm colour if .L3_Bureau; taps .Visu_L3
rounded rectangle at (560,50)-(671,81): text "HealthBox"; alarm colour if .HealthBox; taps .Visu_HealthBox
rounded rectangle at (1180,340)-(1291,371): text "Rolluik neer"; alarm colour if .Rolluik_Voorgevel_Down; taps .Visu_Rolluik_Voorgevel_Down
rounded rectangle at (1180,300)-(1291,331): text "Rolluik op"; alarm colour if .Rolluik_Voorgevel_Up; taps .Visu_Rolluik_Voorgevel_Up
rounded rectangle at (40,240)-(111,271): text "Buiten"; alarm colour if .L1_Oversteek; taps .Visu_Licht_Oversteek
rounded rectangle at (40,620)-(261,651): text "Auto"; alarm colour if AutoMode; taps .Visu_AutoMode
rounded rectangle at (220,50)-(311,81): text "Ontbijtkast"; alarm colour if .L4_Ontbijtkast; taps .Visu_Ontbijtkast
rounded rectangle at (700,120)-(791,151): text "Bijkeuken"; alarm colour if .L6_Bijkeuken; taps .Visu_Bijkeuken
rounded rectangle at (280,500)-(501,531): text "Avond"; taps .Visu_Sfeer_Avond
rounded rectangle at (650,360)-(781,391): text "Living"; alarm colour if .L7_Living; taps .Visu_Licht_Living
22 more shapes without text or variables
*)
